/// machine data that is used through most sequences of the unit (motor speed, axes positions, ...)
TYPE HandlingDataMachine :
STRUCT
  Slowspeed : LREAL;
  Highspeed : LREAL;
END_STRUCT
END_TYPE

(* stored: Version 1.1.0.1
   DUT HandlingDataMachine: Id {c087ff30-5380-440e-9eb1-3a39e0a98c65} *)
